TYPE TcoPlbPaletizator_Control_v_1_x_x EXTENDS TcoCore.TcoStruct:
STRUCT

		ResetOnlyManipulator: BOOL;
		
END_STRUCT
END_TYPE

(* stored: Version 1.1.0.1
   DUT TcoPlbPaletizator_Control_v_1_x_x: Id {c4e611d3-9e15-4525-a940-e072375099e4} *)
